FUNCTION_BLOCK SKILL_PackML (* Reduced PackML skill state machine shared by all skills; completion by Ensures, abort on Invariant violation or watchdog timeout *)
  (* Standard: 61499-2 *)
  (* Version 2.0, 2026-09-27, Project contributors, Filling cell reference model *)
  PACKAGE fillingcell;
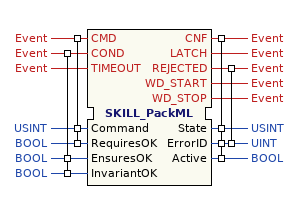
  EVENT_INPUT
    CMD WITH Command, RequiresOK;
    COND WITH EnsuresOK, InvariantOK;
    TIMEOUT;
  END_EVENT
  EVENT_OUTPUT
    CNF WITH State, ErrorID, Active;
    LATCH;
    REJECTED WITH ErrorID;
    WD_START;
    WD_STOP;
  END_EVENT
  VAR_INPUT
    Command : USINT;
    RequiresOK : BOOL;
    EnsuresOK : BOOL;
    InvariantOK : BOOL;
  END_VAR
  VAR_OUTPUT
    State : USINT := 4;
    ErrorID : UINT;
    Active : BOOL;
  END_VAR
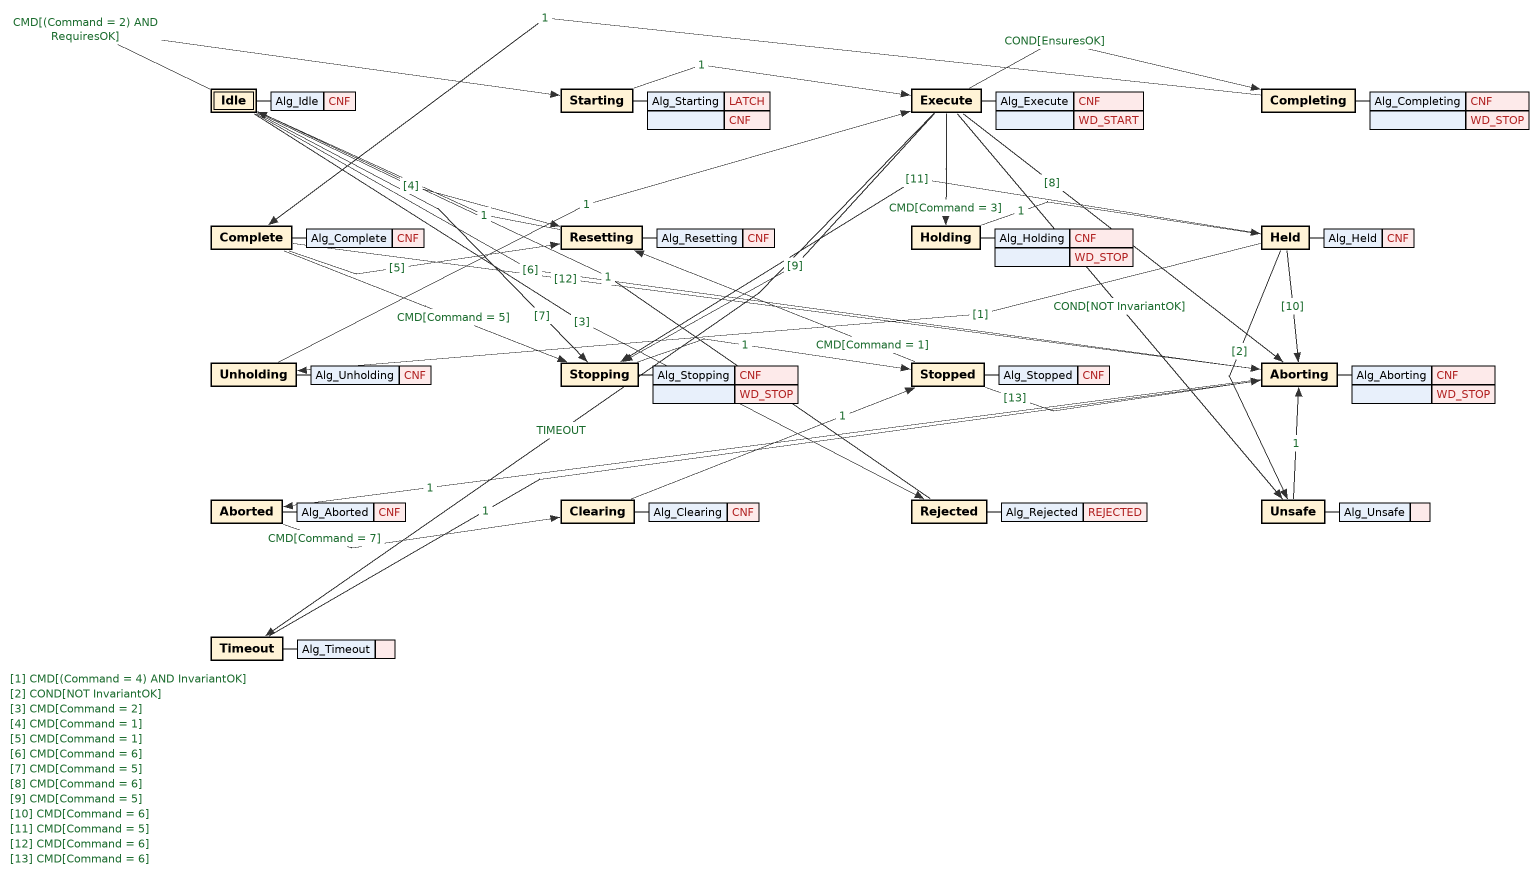
  EC_STATES
    Idle : Alg_Idle -> CNF;
    Starting : Alg_Starting -> LATCH, -> CNF;
    Execute : Alg_Execute -> CNF, -> WD_START;
    Completing : Alg_Completing -> CNF, -> WD_STOP;
    Complete : Alg_Complete -> CNF;
    Resetting : Alg_Resetting -> CNF;
    Holding : Alg_Holding -> CNF, -> WD_STOP;
    Held : Alg_Held -> CNF;
    Unholding : Alg_Unholding -> CNF;
    Stopping : Alg_Stopping -> CNF, -> WD_STOP;
    Stopped : Alg_Stopped -> CNF;
    Aborting : Alg_Aborting -> CNF, -> WD_STOP;
    Aborted : Alg_Aborted -> CNF;
    Clearing : Alg_Clearing -> CNF;
    Rejected : Alg_Rejected -> REJECTED;
    Unsafe : Alg_Unsafe;
    Timeout : Alg_Timeout;
  END_STATES
  EC_TRANSITIONS
    Idle TO Starting := CMD[(Command = 2) AND RequiresOK];
    Idle TO Rejected := CMD[Command = 2];
    Rejected TO Idle := 1;
    Starting TO Execute := 1;
    Execute TO Unsafe := COND[NOT InvariantOK];
    Execute TO Completing := COND[EnsuresOK];
    Execute TO Timeout := TIMEOUT;
    Unsafe TO Aborting := 1;
    Timeout TO Aborting := 1;
    Execute TO Holding := CMD[Command = 3];
    Holding TO Held := 1;
    Held TO Unholding := CMD[(Command = 4) AND InvariantOK];
    Held TO Unsafe := COND[NOT InvariantOK];
    Unholding TO Execute := 1;
    Completing TO Complete := 1;
    Idle TO Resetting := CMD[Command = 1];
    Complete TO Resetting := CMD[Command = 1];
    Stopped TO Resetting := CMD[Command = 1];
    Resetting TO Idle := 1;
    Idle TO Aborting := CMD[Command = 6];
    Idle TO Stopping := CMD[Command = 5];
    Execute TO Aborting := CMD[Command = 6];
    Execute TO Stopping := CMD[Command = 5];
    Held TO Aborting := CMD[Command = 6];
    Held TO Stopping := CMD[Command = 5];
    Complete TO Aborting := CMD[Command = 6];
    Complete TO Stopping := CMD[Command = 5];
    Stopped TO Aborting := CMD[Command = 6];
    Stopping TO Stopped := 1;
    Aborting TO Aborted := 1;
    Aborted TO Clearing := CMD[Command = 7];
    Clearing TO Stopped := 1;
  END_TRANSITIONS
  ALGORITHM Alg_Idle IN ST:
State := 4;
Active := FALSE;
  END_ALGORITHM
  ALGORITHM Alg_Starting IN ST:
State := 3;
Active := FALSE;
ErrorID := 0;
  END_ALGORITHM
  ALGORITHM Alg_Execute IN ST:
State := 6;
Active := TRUE;
  END_ALGORITHM
  ALGORITHM Alg_Completing IN ST:
State := 16;
Active := FALSE;
  END_ALGORITHM
  ALGORITHM Alg_Complete IN ST:
State := 17;
Active := FALSE;
  END_ALGORITHM
  ALGORITHM Alg_Resetting IN ST:
State := 15;
Active := FALSE;
ErrorID := 0;
  END_ALGORITHM
  ALGORITHM Alg_Holding IN ST:
State := 10;
Active := FALSE;
  END_ALGORITHM
  ALGORITHM Alg_Held IN ST:
State := 11;
Active := FALSE;
  END_ALGORITHM
  ALGORITHM Alg_Unholding IN ST:
State := 12;
Active := FALSE;
  END_ALGORITHM
  ALGORITHM Alg_Stopping IN ST:
State := 7;
Active := FALSE;
  END_ALGORITHM
  ALGORITHM Alg_Stopped IN ST:
State := 2;
Active := FALSE;
  END_ALGORITHM
  ALGORITHM Alg_Aborting IN ST:
State := 8;
Active := FALSE;
  END_ALGORITHM
  ALGORITHM Alg_Aborted IN ST:
State := 9;
Active := FALSE;
  END_ALGORITHM
  ALGORITHM Alg_Clearing IN ST:
State := 1;
Active := FALSE;
ErrorID := 0;
  END_ALGORITHM
  ALGORITHM Alg_Rejected IN ST:
ErrorID := 1;
  END_ALGORITHM
  ALGORITHM Alg_Unsafe IN ST:
ErrorID := 2;
  END_ALGORITHM
  ALGORITHM Alg_Timeout IN ST:
ErrorID := 3;
  END_ALGORITHM
END_FUNCTION_BLOCK
